RoboDK station: Exercises1_2.rdk

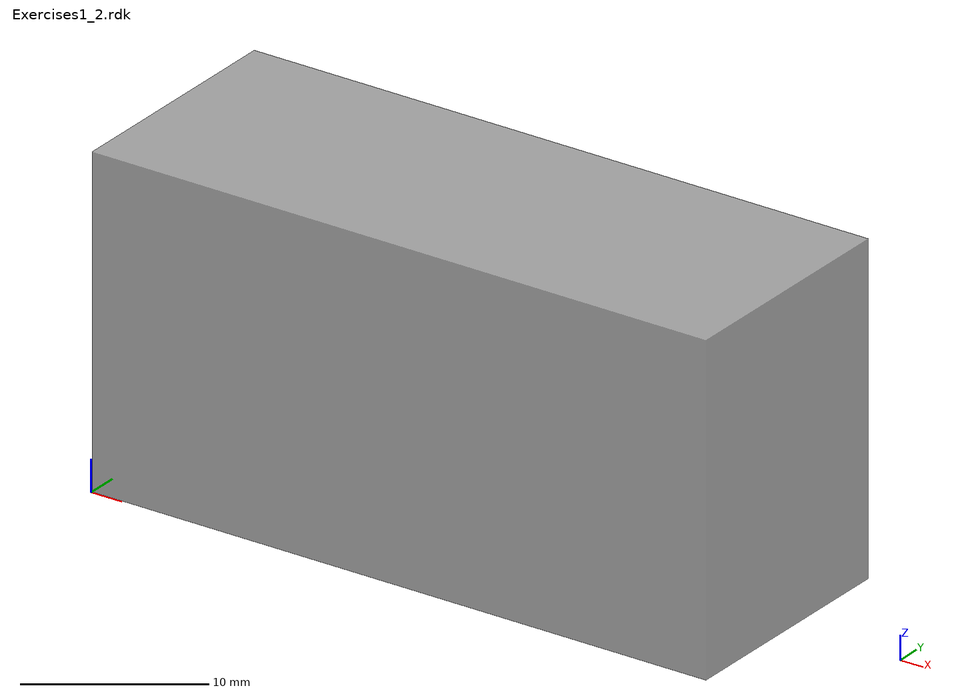
[picture v0: the station drawn from its stored meshes, robots at their saved joint values, targets as dots, program paths as lines]
Station World (saved by RoboDK 5.8.0). Poses are relative to the parent item; angles as X-Y-Z fixed-axis rotations.
  - frame A-Frame at (0, 0, 0) mm
  - frame B-Frame at (0, 0, 0) mm
    - object myBrick at (0, 0, 0) mm, size 39.7 x 15 x 20 mm, geometry from myBrick.stl
